FUNCTION_BLOCK Achsfreigabe
VAR_INPUT
END_VAR
VAR_OUTPUT
END_VAR
VAR
END_VAR

// NETWORK 1

END_FUNCTION_BLOCK

(* stored: Version 1.1.0.1, ProductVersion 3.1.4024.4
   POU Achsfreigabe: Id {fbb82708-2c4f-4e89-9571-dc48c49d61a7}, SpecialFunc None *)
